(* PLC project Unnamed, Unknown Unnamed 1 *)
(* stored: creationDateTime 2025-10-22T19:37:31, modificationDateTime 2025-10-24T02:02:38 *)

PROGRAM plc_controller
  VAR
    In_Start_Stop AT %IX0.2 : BOOL;
    In_Temp_Up AT %IX0.0 : BOOL;
    In_Temp_Down AT %IX0.1 : BOOL;
    Out_Status_LED AT %QX0.7 : BOOL;
    Out_Display_LED0 AT %QX0.6 : BOOL;
    Out_Display_LED1 AT %QX0.5 : BOOL;
    Out_Display_LED2 AT %QX0.4 : BOOL;
    Out_Display_LED3 AT %QX0.3 : BOOL;
    Out_Display_LED4 AT %QX0.2 : BOOL;
    Out_Display_LED5 AT %QX0.1 : BOOL;
  END_VAR
  VAR
    Heating_On : BOOL := FALSE;
    Temp_Setting : INT;
    MAX_TEMP_SETTING : INT := 10;  (* CONSTANT describes the maximum temperature setting *)
    R_TRIG0 : R_TRIG;
    CTUD0 : CTUD;
  END_VAR
  VAR  (* added by the conversion: wires and edge detectors of the diagram *)
    _NOT21_OUT : BOOL;
    R_TRIG1 : R_TRIG;
    R_TRIG2 : R_TRIG;
    _NOT136_OUT : BOOL;
  END_VAR

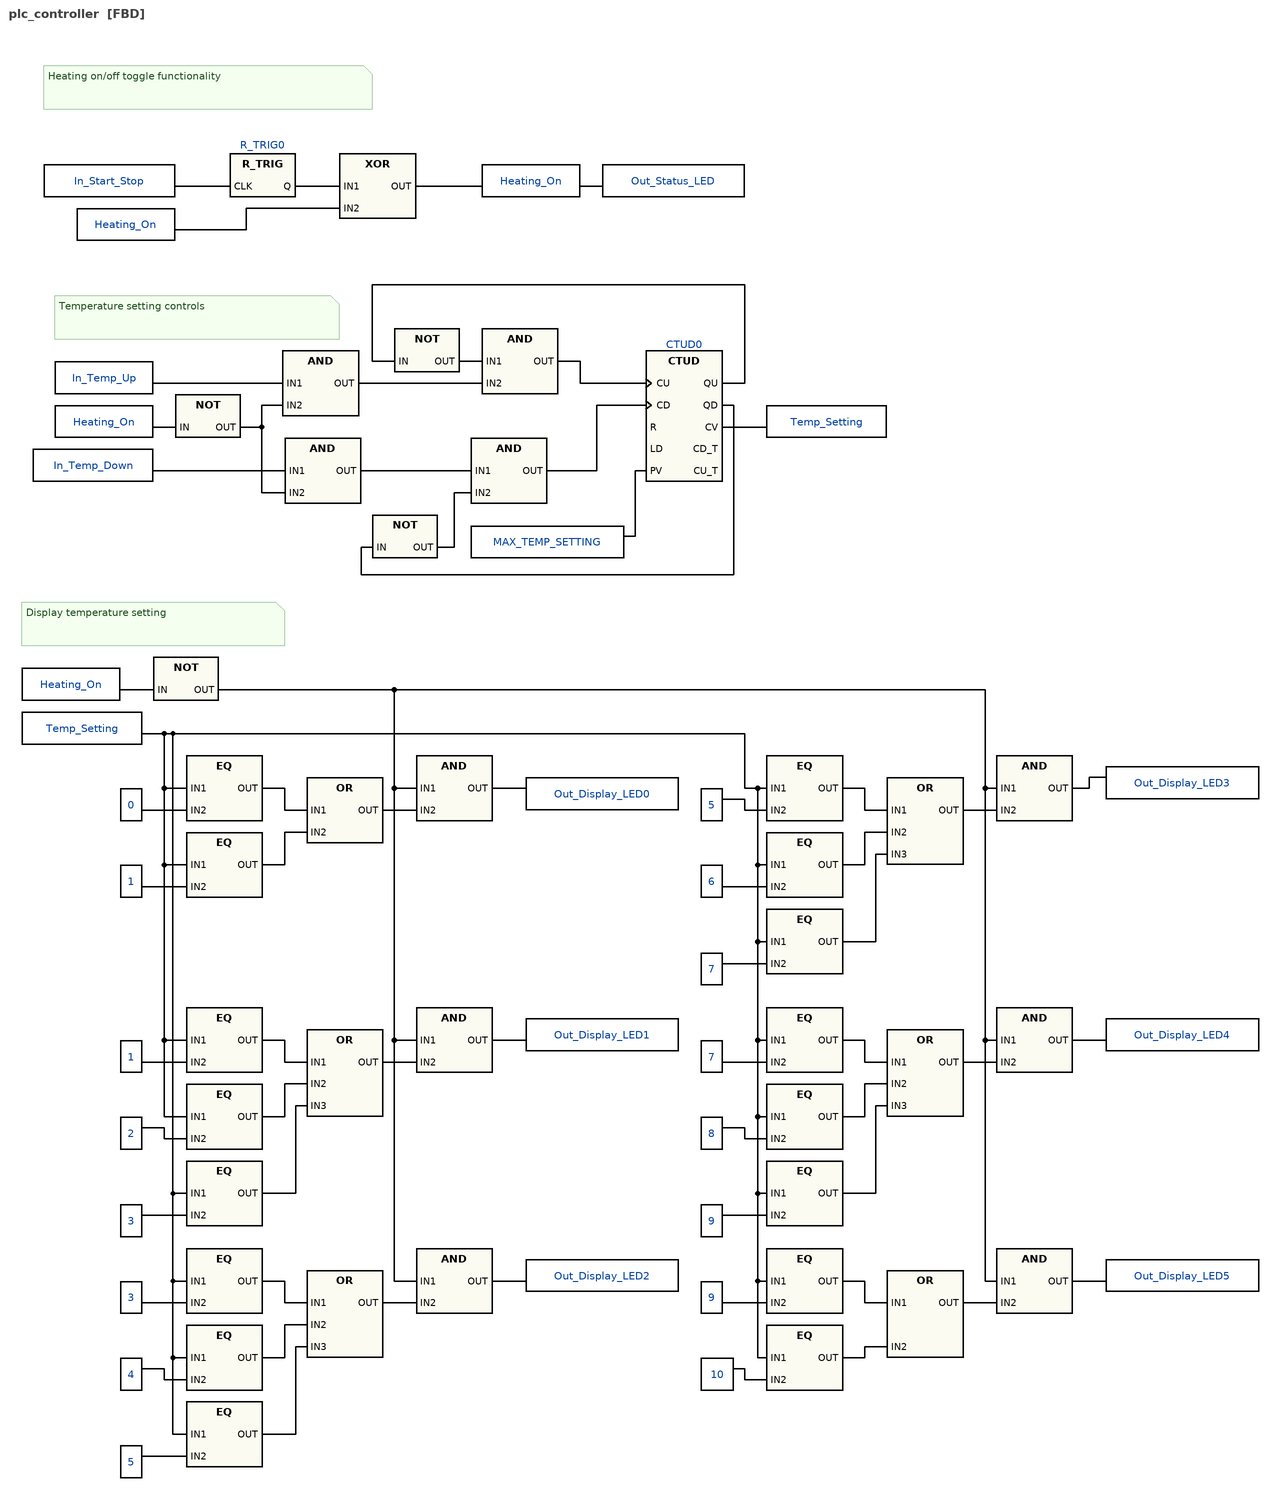
(* FBD diagram, written out as Structured Text *)
(* Heating on/off toggle functionality *)
(* Temperature setting controls *)
_NOT21_OUT := NOT Heating_On;
R_TRIG1(CLK := NOT CTUD0.QU AND In_Temp_Up AND _NOT21_OUT);
R_TRIG2(CLK := In_Temp_Down AND _NOT21_OUT AND NOT CTUD0.QD);
CTUD0(CU := R_TRIG1.Q, CD := R_TRIG2.Q, PV := MAX_TEMP_SETTING);
Temp_Setting := CTUD0.CV;
R_TRIG0(CLK := In_Start_Stop);
Heating_On := R_TRIG0.Q XOR Heating_On;
Out_Status_LED := Heating_On;
(* Display temperature setting *)
_NOT136_OUT := NOT Heating_On;
Out_Display_LED0 := _NOT136_OUT AND (Temp_Setting = 0 OR Temp_Setting = 1);
Out_Display_LED3 := _NOT136_OUT AND (Temp_Setting = 5 OR Temp_Setting = 6 OR Temp_Setting = 7);
Out_Display_LED1 := _NOT136_OUT AND (Temp_Setting = 1 OR Temp_Setting = 2 OR Temp_Setting = 3);
Out_Display_LED4 := _NOT136_OUT AND (Temp_Setting = 7 OR Temp_Setting = 8 OR Temp_Setting = 9);
Out_Display_LED2 := _NOT136_OUT AND (Temp_Setting = 3 OR Temp_Setting = 4 OR Temp_Setting = 5);
Out_Display_LED5 := _NOT136_OUT AND (Temp_Setting = 9 OR Temp_Setting = 10);
END_PROGRAM

CONFIGURATION Config0
  RESOURCE Res0 ON PLC
    TASK task0(INTERVAL := T#20ms, PRIORITY := 0);
    PROGRAM instance0 WITH task0 : plc_controller;
  END_RESOURCE
END_CONFIGURATION
